// TIA Portal project "LIFT PROJECT" (V19)

(* hardware
DEVICE "S7-1200 station_1"  S7-1200 Station
   slot 0: "Rack_0"  S7-1200 Rack  Rack  V1.0
   slot 1: "PLC_1"  CPU 1211C AC/DC/Rly  6ES7 211-1BE40-0XB0  V4.6
*)

// ===== PLC "PLC_1"  CPU 1211C AC/DC/Rly =====

VAR_GLOBAL   // PLC tag table "Default tag table"
   "STOP PB" AT %I5.0 : Bool;
   "GET LIFT 0" AT %I5.1 : Bool;
   "GET LIFT 1" AT %I5.2 : Bool;
   "GET LIFT 2" AT %I5.3 : Bool;
   "GET LIFT 3" AT %I5.4 : Bool;
   "GROUND FLOOR" AT %I5.5 : Bool;
   "1ST FLOOR" AT %I5.6 : Bool;
   "2ND FLOOR" AT %I5.7 : Bool;
   "3RD FLOOR" AT %I6.0 : Bool;
   "GROUND FLOOR SLOW" AT %I6.1 : Bool;
   "GROUND FLOOR SENSOR" AT %I6.2 : Bool;
   "1ST FLOOR SLOW" AT %I6.3 : Bool;
   "1ST FLOOR SLOW 2" AT %I6.4 : Bool;
   "1ST FLOOR SENSOR" AT %I6.5 : Bool;
   "2ND FLOOR SLOW" AT %I6.6 : Bool;
   "2ND FLOOR SLOW 2" AT %I6.7 : Bool;
   "2ND FLOOR SENSOR" AT %I7.0 : Bool;
   "3RD FLOOR SLOW" AT %I7.1 : Bool;
   "3RD FLOOR SENSOR" AT %I7.2 : Bool;
   "START PB" AT %I7.3 : Bool;
   "Elevator UP" AT %Q0.0 : Bool;
   "Elevator DOWN" AT %Q0.1 : Bool;
   "Elevator SLOW" AT %Q0.2 : Bool;
   "SYSTEM_ON" AT %Q0.3 : Bool;
   "TARGET FLOOR" AT %MW0 : Int;
   "CURRENT FLOOR" AT %MW2 : Int;
   "Tag_1" AT %MW4 : Int;
   "Tag_2" AT %MW6 : Int;
   "Tag_3" AT %MW8 : Int;
   "Tag_4" AT %MW10 : Int;
END_VAR

// folder: System blocks/Program resources

DATA_BLOCK "IEC_Timer_0_DB_1"   // DB1
{ S7_Optimized_Access := 'TRUE' }
AUTHOR : Simatic
FAMILY : IEC
NAME : IEC_TMR
VERSION : 1.0
// stored: InstanceOfName IEC_TIMER
"IEC_TIMER"
BEGIN
END_DATA_BLOCK

DATA_BLOCK "IEC_Timer_0_DB_2"   // DB2
{ S7_Optimized_Access := 'TRUE' }
AUTHOR : Simatic
FAMILY : IEC
NAME : IEC_TMR
VERSION : 1.0
// stored: InstanceOfName IEC_TIMER
"IEC_TIMER"
BEGIN
END_DATA_BLOCK

DATA_BLOCK "IEC_Timer_0_DB_3"   // DB3
{ S7_Optimized_Access := 'TRUE' }
AUTHOR : Simatic
FAMILY : IEC
NAME : IEC_TMR
VERSION : 1.0
// stored: InstanceOfName IEC_TIMER
"IEC_TIMER"
BEGIN
END_DATA_BLOCK

DATA_BLOCK "IEC_Timer_0_DB_4"   // DB4
{ S7_Optimized_Access := 'TRUE' }
AUTHOR : Simatic
FAMILY : IEC
NAME : IEC_TMR
VERSION : 1.0
// stored: InstanceOfName IEC_TIMER
"IEC_TIMER"
BEGIN
END_DATA_BLOCK

DATA_BLOCK "IEC_Timer_0_DB"   // DB5
{ S7_Optimized_Access := 'TRUE' }
AUTHOR : Simatic
FAMILY : IEC
NAME : IEC_TMR
VERSION : 1.0
// stored: InstanceOfName IEC_TIMER
"IEC_TIMER"
BEGIN
END_DATA_BLOCK

// folder: (top level)

FUNCTION "MHJ-PLC-Lab-Function-S71200" : Void   // FC9000, SCL
{ S7_Optimized_Access := 'TRUE' }
VERSION : 0.1
   VAR_TEMP
      rdTimeReturn : Int;
      outputTime : DTL;
      SyncVal : Byte;
      forVal : Int;
      forVal_2 : Int;
      Value : Byte;
   END_VAR
   VAR CONSTANT
      CompVal : Byte := 16#34;
      Value_01 : Byte := 16#11;
      Value_01_DW : DWord := 16#A165_D992;
      Value_02_DW : DWord := 16#58BE_4401;
   END_VAR
BEGIN

   #Value:=PEEK(area := 16#82,
        dbNumber := 0,
        byteOffset := 511);
   #Value := #Value + 1;

   POKE(area := 16#82,
        dbNumber := 0,
        byteOffset := 511,
        value := #Value);

   POKE(area:=16#81,
        dbNumber:=0,
        byteOffset:=1016,
        value:=#Value_01_DW);
   POKE(area := 16#81,
        dbNumber := 0,
        byteOffset := 1020,
        value := #Value_02_DW);

   POKE(area := 16#81,
        dbNumber := 0,
        byteOffset := 511,
        value := B#16#00);

   FOR #forVal := 0 TO 120 DO
       FOR #forVal_2:=0 TO 10 DO
           #rdTimeReturn:=RD_SYS_T(#outputTime);
           #rdTimeReturn := WR_SYS_T(#outputTime);
           #rdTimeReturn := RD_SYS_T(#outputTime);
           #rdTimeReturn := WR_SYS_T(#outputTime);
       END_FOR;
       #SyncVal:= PEEK(area := 16#81,
                      dbNumber := 0,
                      byteOffset := 511);
       IF #SyncVal = #CompVal THEN
          GOTO M_1;
       END_IF;
   END_FOR;
   RETURN;

   M_1:
   POKE(area := 16#81,
        dbNumber := 0,
        byteOffset := 511,
        value := B#16#0);
END_FUNCTION

ORGANIZATION_BLOCK "Main"   // OB1, LAD, ProgramCycle
TITLE = "Main Program Sweep (Cycle)"
{ S7_Optimized_Access := 'TRUE' }
VERSION : 0.1
   VAR_INPUT
      Initial_Call : Bool;   // Initial call of this OB
      Remanence : Bool;   // =True, if remanent data are available
   END_VAR
BEGIN

REGION Network 1
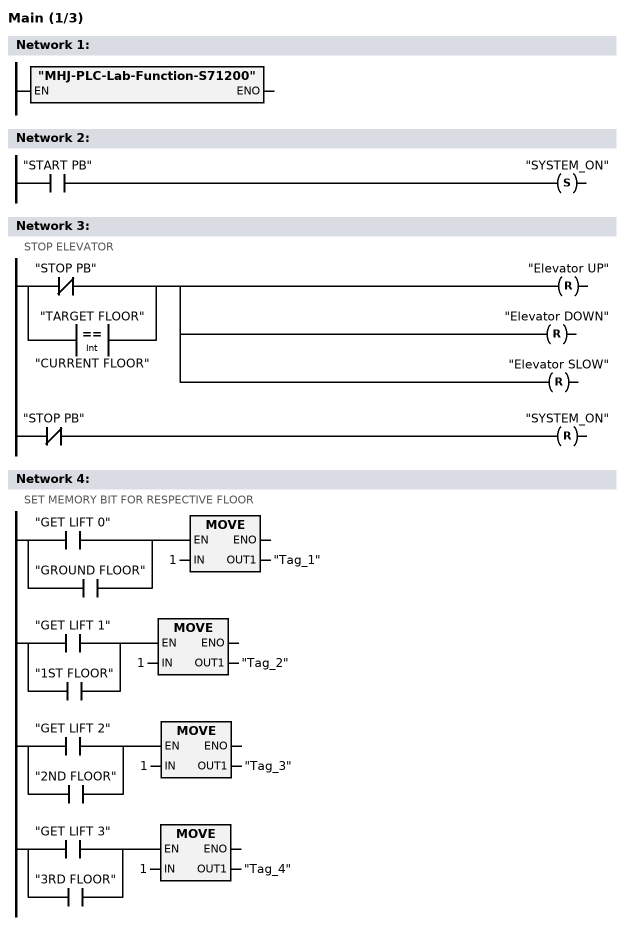
   RUNG wire#powerrail
      "MHJ-PLC-Lab-Function-S71200"()
   END_RUNG
   // the same network as SCL:
   "MHJ-PLC-Lab-Function-S71200"();
END_REGION

REGION Network 2
   RUNG wire#powerrail
      Contact( "START PB" )
      S_Coil( "SYSTEM_ON" )
   END_RUNG
   // the same network as SCL:
   IF "START PB" THEN "SYSTEM_ON" := TRUE; END_IF;
END_REGION

REGION Network 3
   // STOP ELEVATOR
   RUNG wire#powerrail
      I_Contact( "STOP PB" )
      wire#w1
      R_Coil( "Elevator UP" )
   END_RUNG
   RUNG wire#powerrail
      { S7_Templates := "SrcType := Int" } EQ_Contact(in1 := "TARGET FLOOR", in2 := "CURRENT FLOOR")
   END_RUNG wire#w1
   RUNG wire#w1
      R_Coil( "Elevator DOWN" )
   END_RUNG
   RUNG wire#w1
      R_Coil( "Elevator SLOW" )
   END_RUNG
   RUNG wire#powerrail
      I_Contact( "STOP PB" )
      R_Coil( "SYSTEM_ON" )
   END_RUNG
   // the same network as SCL:
   IF NOT "STOP PB" OR ("TARGET FLOOR" = "CURRENT FLOOR") THEN
       "Elevator UP" := FALSE;
       "Elevator DOWN" := FALSE;
       "Elevator SLOW" := FALSE;
   END_IF;
   IF NOT "STOP PB" THEN "SYSTEM_ON" := FALSE; END_IF;
END_REGION

REGION Network 4
   // SET MEMORY BIT FOR RESPECTIVE FLOOR
   RUNG wire#powerrail
      Contact( "GET LIFT 0" )
      wire#w1
      Move(in := 1, out1 => "Tag_1")
   END_RUNG
   RUNG wire#powerrail
      Contact( "GROUND FLOOR" )
   END_RUNG wire#w1
   RUNG wire#powerrail
      Contact( "GET LIFT 1" )
      wire#w2
      Move(in := 1, out1 => "Tag_2")
   END_RUNG
   RUNG wire#powerrail
      Contact( "1ST FLOOR" )
   END_RUNG wire#w2
   RUNG wire#powerrail
      Contact( "GET LIFT 2" )
      wire#w3
      Move(in := 1, out1 => "Tag_3")
   END_RUNG
   RUNG wire#powerrail
      Contact( "2ND FLOOR" )
   END_RUNG wire#w3
   RUNG wire#powerrail
      Contact( "GET LIFT 3" )
      wire#w4
      Move(in := 1, out1 => "Tag_4")
   END_RUNG
   RUNG wire#powerrail
      Contact( "3RD FLOOR" )
   END_RUNG wire#w4
   // the same network as SCL:
   IF "GET LIFT 0" OR "GROUND FLOOR" THEN "Tag_1" := 1; END_IF;
   IF "GET LIFT 1" OR "1ST FLOOR" THEN "Tag_2" := 1; END_IF;
   IF "GET LIFT 2" OR "2ND FLOOR" THEN "Tag_3" := 1; END_IF;
   IF "GET LIFT 3" OR "3RD FLOOR" THEN "Tag_4" := 1; END_IF;
END_REGION

REGION Network 5
   // MOVE TARGET FLOOR NUMBER
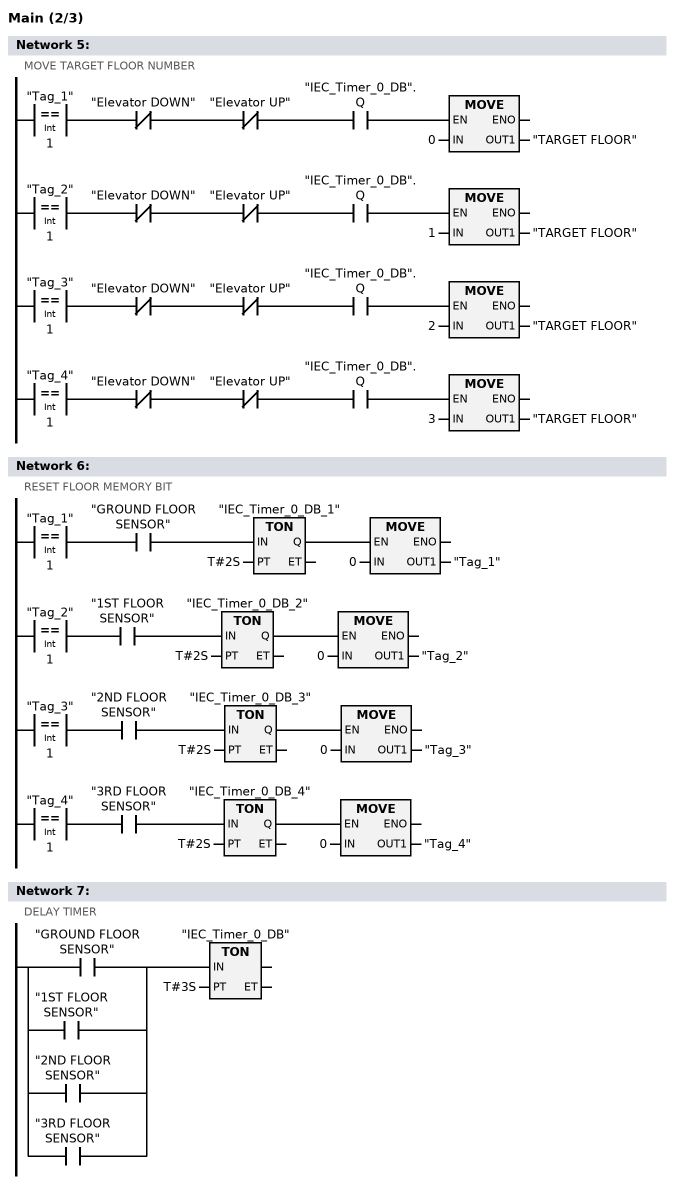
   RUNG wire#powerrail
      { S7_Templates := "SrcType := Int" } EQ_Contact(in1 := "Tag_1", in2 := 1)
      I_Contact( "Elevator DOWN" )
      I_Contact( "Elevator UP" )
      Contact( "IEC_Timer_0_DB".Q )
      Move(in := 0, out1 => "TARGET FLOOR")
   END_RUNG
   RUNG wire#powerrail
      { S7_Templates := "SrcType := Int" } EQ_Contact(in1 := "Tag_2", in2 := 1)
      I_Contact( "Elevator DOWN" )
      I_Contact( "Elevator UP" )
      Contact( "IEC_Timer_0_DB".Q )
      Move(in := 1, out1 => "TARGET FLOOR")
   END_RUNG
   RUNG wire#powerrail
      { S7_Templates := "SrcType := Int" } EQ_Contact(in1 := "Tag_3", in2 := 1)
      I_Contact( "Elevator DOWN" )
      I_Contact( "Elevator UP" )
      Contact( "IEC_Timer_0_DB".Q )
      Move(in := 2, out1 => "TARGET FLOOR")
   END_RUNG
   RUNG wire#powerrail
      { S7_Templates := "SrcType := Int" } EQ_Contact(in1 := "Tag_4", in2 := 1)
      I_Contact( "Elevator DOWN" )
      I_Contact( "Elevator UP" )
      Contact( "IEC_Timer_0_DB".Q )
      Move(in := 3, out1 => "TARGET FLOOR")
   END_RUNG
   // the same network as SCL:
   IF ("Tag_1" = 1) AND NOT "Elevator DOWN" AND NOT "Elevator UP" AND "IEC_Timer_0_DB".Q THEN
       "TARGET FLOOR" := 0;
   END_IF;
   IF ("Tag_2" = 1) AND NOT "Elevator DOWN" AND NOT "Elevator UP" AND "IEC_Timer_0_DB".Q THEN
       "TARGET FLOOR" := 1;
   END_IF;
   IF ("Tag_3" = 1) AND NOT "Elevator DOWN" AND NOT "Elevator UP" AND "IEC_Timer_0_DB".Q THEN
       "TARGET FLOOR" := 2;
   END_IF;
   IF ("Tag_4" = 1) AND NOT "Elevator DOWN" AND NOT "Elevator UP" AND "IEC_Timer_0_DB".Q THEN
       "TARGET FLOOR" := 3;
   END_IF;
END_REGION

REGION Network 6
   // RESET FLOOR MEMORY BIT
   "IEC_Timer_0_DB_1".TON(IN := ("Tag_1" = 1) AND "GROUND FLOOR SENSOR", PT := T#2S);
   IF "IEC_Timer_0_DB_1".Q THEN "Tag_1" := 0; END_IF;
   "IEC_Timer_0_DB_2".TON(IN := ("Tag_2" = 1) AND "1ST FLOOR SENSOR", PT := T#2S);
   IF "IEC_Timer_0_DB_2".Q THEN "Tag_2" := 0; END_IF;
   "IEC_Timer_0_DB_3".TON(IN := ("Tag_3" = 1) AND "2ND FLOOR SENSOR", PT := T#2S);
   IF "IEC_Timer_0_DB_3".Q THEN "Tag_3" := 0; END_IF;
   "IEC_Timer_0_DB_4".TON(IN := ("Tag_4" = 1) AND "3RD FLOOR SENSOR", PT := T#2S);
   IF "IEC_Timer_0_DB_4".Q THEN "Tag_4" := 0; END_IF;
END_REGION

REGION Network 7
   // DELAY TIMER
   "IEC_Timer_0_DB".TON(IN := "GROUND FLOOR SENSOR" OR "1ST FLOOR SENSOR" OR "2ND FLOOR SENSOR" OR "3RD FLOOR SENSOR",
                        PT := T#3S);
END_REGION

REGION Network 8
   // MOVE CURRENT FLOOR IN DATA REGISTER
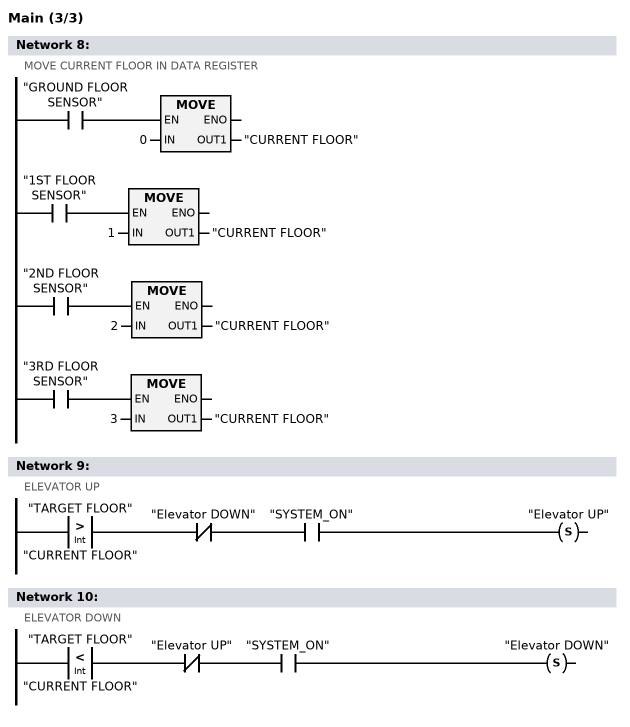
   RUNG wire#powerrail
      Contact( "GROUND FLOOR SENSOR" )
      Move(in := 0, out1 => "CURRENT FLOOR")
   END_RUNG
   RUNG wire#powerrail
      Contact( "1ST FLOOR SENSOR" )
      Move(in := 1, out1 => "CURRENT FLOOR")
   END_RUNG
   RUNG wire#powerrail
      Contact( "2ND FLOOR SENSOR" )
      Move(in := 2, out1 => "CURRENT FLOOR")
   END_RUNG
   RUNG wire#powerrail
      Contact( "3RD FLOOR SENSOR" )
      Move(in := 3, out1 => "CURRENT FLOOR")
   END_RUNG
   // the same network as SCL:
   IF "GROUND FLOOR SENSOR" THEN "CURRENT FLOOR" := 0; END_IF;
   IF "1ST FLOOR SENSOR" THEN "CURRENT FLOOR" := 1; END_IF;
   IF "2ND FLOOR SENSOR" THEN "CURRENT FLOOR" := 2; END_IF;
   IF "3RD FLOOR SENSOR" THEN "CURRENT FLOOR" := 3; END_IF;
END_REGION

REGION Network 9
   // ELEVATOR UP
   RUNG wire#powerrail
      { S7_Templates := "SrcType := Int" } GT_Contact(in1 := "TARGET FLOOR", in2 := "CURRENT FLOOR")
      I_Contact( "Elevator DOWN" )
      Contact( "SYSTEM_ON" )
      S_Coil( "Elevator UP" )
   END_RUNG
   // the same network as SCL:
   IF ("TARGET FLOOR" > "CURRENT FLOOR") AND NOT "Elevator DOWN" AND "SYSTEM_ON" THEN
       "Elevator UP" := TRUE;
   END_IF;
END_REGION

REGION Network 10
   // ELEVATOR DOWN
   RUNG wire#powerrail
      { S7_Templates := "SrcType := Int" } LT_Contact(in1 := "TARGET FLOOR", in2 := "CURRENT FLOOR")
      I_Contact( "Elevator UP" )
      Contact( "SYSTEM_ON" )
      S_Coil( "Elevator DOWN" )
   END_RUNG
   // the same network as SCL:
   IF ("TARGET FLOOR" < "CURRENT FLOOR") AND NOT "Elevator UP" AND "SYSTEM_ON" THEN
       "Elevator DOWN" := TRUE;
   END_IF;
END_REGION
END_ORGANIZATION_BLOCK